(* CoDeSys 2.3.10.0 project: CXxxxx.pro *)
(* Libraries: STANDARD.LIB 5.6.98 13:03:02, TcBase.lib 14.5.09 13:14:08, TcSystem.lib 9.3.10 11:21:30, TcUtilities.lib 7.4.10 10:22:08 *)

(* Task configuration *)
TASK Standard (PRIORITY := 0, INTERVAL := T#10ms);
	MAIN
END_TASK

(* Global variable list: Global_Persistent *)
VAR_GLOBAL PERSISTENT
(* Zmienne przechowywane na karcie CF *)
	CF_Persistent_Bool:		BOOL;
	CF_Persistent_Integer:	INT;
	CF_Persistent_String:	STRING;
	CF_Persistent_Real:		REAL;
END_VAR

(* Global variable list: Global_Variables *)
VAR_GLOBAL
(*Zmienne przechowywane w pamieci NOV DP-RAM*)
	Persistent_Bool		AT %Q*:BOOL;
	Persistent_Integer	AT %Q*:INT;
	Persistent_String		AT %Q*:STRING;
	Persistent_Real		AT %Q*:REAL;
END_VAR

(* Global variable list: TwinCAT_Configuration *)
(* Generated automatically by TwinCAT - (read only) *)
VAR_CONFIG
	.Persistent_Bool AT %QX87.0 : BOOL;	(*  ~ {LinkedWith:TIID^Device 4 (NOV/DP-RAM)^Outputs^Persistent_Bool} *)
	.Persistent_Integer AT %QB0 : INT;	(*  ~ {LinkedWith:TIID^Device 4 (NOV/DP-RAM)^Outputs^Persistent_Integer} *)
	.Persistent_String AT %QB2 : STRING(80);	(*  ~ {LinkedWith:TIID^Device 4 (NOV/DP-RAM)^Outputs^Persistent_String} *)
	.Persistent_Real AT %QB83 : REAL;	(*  ~ {LinkedWith:TIID^Device 4 (NOV/DP-RAM)^Outputs^Persistent_Real} *)
END_VAR

(* POU MAIN, CFC *)
PROGRAM MAIN
VAR
	fbPersistent: FB_Persistent;
	bWrite:BOOL;
	tCzas: TIME:=T#2h;
	bBusy: BOOL;
	bErr: BOOL;
	udErrid: UDINT;
	ctu1: CTU;
END_VAR
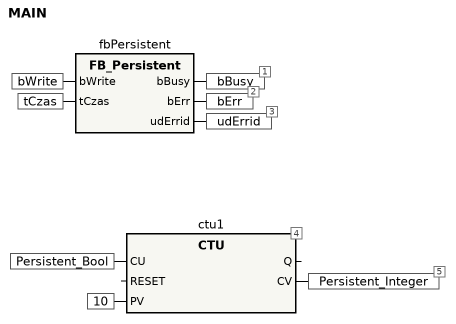
_CFC_ (* Continuous Function Chart, elements in execution order *)
#0 fbPersistent:FB_Persistent(bWrite: bWrite, tCzas: tCzas)
#1 bBusy <= #0.bBusy
#2 bErr <= #0.bErr
#3 udErrid <= #0.udErrid
#4 ctu1:CTU(CU: Persistent_Bool, RESET: -, PV: 10)
#5 Persistent_Integer <= #4.CV
_END_CFC_
(* the same logic as Structured Text *)
fbPersistent(bWrite := bWrite, tCzas := tCzas);
bBusy := fbPersistent.bBusy;
bErr := fbPersistent.bErr;
udErrid := fbPersistent.udErrid;
ctu1(CU := Persistent_Bool, PV := 10);
Persistent_Integer := ctu1.CV;
END_PROGRAM

(* POU FB_Persistent, FBD *)
FUNCTION_BLOCK FB_Persistent

(*********************************************************************************************************************************)
(*								Beckhoff Automation Poland									*)
(* 									FB_Persistent 	v1.2									*)
(* 										2.8.2010											*)
(* 					Blok funkcyjny zapisujący zmienne typu persistent na karcie CF CX-a				*)
(* 				Konieczne jest dodanie biblioteki TcUtilities.lib, TcSystem.lib oraz TcBase.lib			*)
(*___________________________________________________________________________________________*)

VAR_INPUT
	bWrite:BOOL;			(*Zapis na rozkaz *)
	tCzas: TIME:=T#1h;		(*Czestotliwosc zapisu na karte CF*)
END_VAR
VAR_OUTPUT
	bBusy: BOOL;
	bErr: BOOL;
	udErrid: UDINT;
END_VAR
VAR
	fbWritePersistentData: FB_WritePersistentData;
	t1: TON;
END_VAR
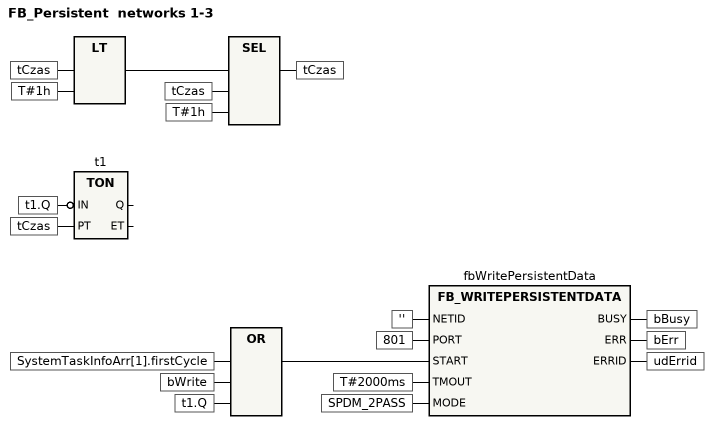
_FBD_ (* Function Block Diagram *)
NETWORK 1 (* Comment: Zabezpieczenie karty - czestotliwosc zapisu nie moze byc mniejsza niz godzina *)
	SEL(LT(tCzas, T#1h), tCzas, T#1h) => tCzas
NETWORK 2 (* Comment: Wyzwalanie zapisu *)
	t1:TON(IN: NOT t1.Q, PT: tCzas)
NETWORK 3 (* Comment: Blok zapisu *)
	fbWritePersistentData:FB_WRITEPERSISTENTDATA(NETID: '', PORT: 801, START: OR(SystemTaskInfoArr[1].firstCycle, bWrite, t1.Q), TMOUT: T#2000ms, MODE: SPDM_2PASS, ERR => bErr, ERRID => udErrid) => bBusy
_END_FBD_
(* the same logic as Structured Text *)
(* Network 1: Comment: Zabezpieczenie karty - czestotliwosc zapisu nie moze byc mniejsza niz godzina *)
tCzas := SEL(tCzas < T#1h, tCzas, T#1h);
(* Network 2: Comment: Wyzwalanie zapisu *)
t1(IN := NOT t1.Q, PT := tCzas);
(* Network 3: Comment: Blok zapisu *)
fbWritePersistentData(NETID := '', PORT := 801, START := SystemTaskInfoArr[1].firstCycle OR bWrite OR t1.Q, TMOUT := T#2000ms, MODE := SPDM_2PASS);
bErr := fbWritePersistentData.ERR;
udErrid := fbWritePersistentData.ERRID;
bBusy := fbWritePersistentData.BUSY;
END_FUNCTION_BLOCK
